Yaskawa INFORM job: R1_W45-48(90,0)KM-OK.JBI

/JOB
//NAME R1_W45-48(90,0)KM-OK
///FOLDERNAME KRIS-SCIANA
//POS
///NPOS 86,86,0,6,0,0
///TOOL 0
///POSTYPE PULSE
///PULSE
C00000=614,-36100,-109393,-1002,105622,76266
C00001=-30112,-127063,-118472,9266,74977,65479
C00002=-146783,-41222,-44528,14508,92298,23932
C00003=-177758,-18432,-24897,15900,96897,12902
C00004=-166847,35431,29185,16026,89350,15768
C00005=-166321,37118,32341,15327,88247,16677
C00006=-166321,37589,33997,15328,87496,16584
C00007=-166321,37118,32341,15327,88247,16677
C00008=-171699,4841,-760,15279,92918,15369
C00009=-170835,-35200,-22324,18799,58263,10772
C00010=-166066,-33100,-15421,17623,54185,12058
C00011=-165910,-32536,-14743,17588,54031,12098
C00012=-165593,-31712,-14199,17442,54048,12239
C00013=-167025,-37605,-22579,17571,56389,12034
C00014=-161139,-1958,-5557,939,83085,16350
C00015=-160390,25614,20531,865,81188,16590
C00016=-160390,25904,21696,866,80621,16587
C00017=-160640,27890,23636,893,80451,16499
C00018=-160390,25457,19886,865,81505,16593
C00019=-160390,25655,20697,865,81108,16591
C00020=-160390,25965,21925,866,80512,16587
C00021=-160390,25906,21695,866,80622,16587
C00022=-160724,27768,23517,901,80463,16471
C00023=-160390,25446,19834,865,81532,16594
C00024=-165643,13675,12551,10985,79337,20135
C00025=-167674,10013,12505,14753,77464,21361
C00026=-167674,10387,13747,14782,76911,21293
C00027=-167674,10317,13522,14776,77011,21304
C00028=-167700,12673,15637,14783,76929,21284
C00029=-167674,9804,11798,14735,77782,21397
C00030=-161667,10120,9793,4034,79193,25528
C00031=-160919,6459,2756,3926,81599,25861
C00032=-171280,-20527,-2481,28534,71438,-2255
C00033=-169873,-15007,4957,28696,69425,-2217
C00034=-167060,-14489,6711,28588,67760,-1526
C00035=-167060,-13749,8427,28718,67162,-1682
C00036=-167060,-14037,7762,28667,67393,-1622
C00037=-166465,-12361,9034,28595,67262,-1417
C00038=-167060,-14860,5838,28526,68066,-1445
C00039=-165078,-24102,-3856,28103,68483,-543
C00040=-174496,-24787,-5330,32767,69285,-4466
C00041=-172819,-19212,1769,32913,67371,-4356
C00042=-172173,-16914,4714,32988,66590,-4329
C00043=-171876,-16211,5234,32949,66511,-4228
C00044=-171876,-15504,6876,33099,65965,-4402
C00045=-171876,-15676,6480,33063,66097,-4360
C00046=-171337,-14366,7462,32993,65949,-4178
C00047=-171876,-15676,6480,33063,66097,-4360
C00048=-161265,-34405,-11426,23449,56557,2204
C00049=-165693,-30942,-7306,24884,57138,447
C00050=-166684,-37324,-14511,24847,58482,354
C00051=-186406,-34667,3928,73065,39460,38715
C00052=-184274,-31936,5659,72637,38187,39290
C00053=-183330,-31185,5556,72054,37725,39763
C00054=-184413,-32109,5553,72669,38270,39251
C00055=-183286,-31712,4384,71496,37848,40087
C00056=-183300,-30553,6129,72089,37695,39749
C00057=-184249,-31903,5681,72632,38172,39297
C00058=-186379,-34635,3948,73060,39445,38722
C00059=-168921,11501,9513,23787,62861,33812
C00060=-168977,15186,12854,23838,62728,33759
C00061=-168277,18170,15265,23592,62571,34011
C00062=-168933,14800,11613,23711,63235,33889
C00063=-168567,15646,14088,23805,62129,33795
C00064=-174514,12133,12884,25971,62948,31524
C00065=-174025,9736,7933,25443,64442,32081
C00066=-174066,6103,4745,25437,64541,32088
C00067=-165320,32292,30686,7449,75670,58759
C00068=-160580,40426,45052,9326,72009,60014
C00069=-168555,20447,28596,16427,68120,-19338
C00070=-168800,19872,28619,16504,67872,-19465
C00071=-157617,30618,37910,-7922,59943,61772
C00072=-157851,30496,37789,-7848,59932,61681
C00073=-159523,23474,32009,-7611,56187,61651
C00074=-170844,18084,26765,-2961,55783,56770
C00075=-171318,17827,26691,-2775,55680,56585
C00076=-172522,13662,24258,-755,52693,56042
C00077=-172766,11273,22657,-34,51599,55901
C00078=-172411,10671,22440,-198,51422,56051
C00079=-172687,-7816,-30,-66,55750,55932
C00080=-179212,-27838,-26858,-4490,80741,54483
C00081=-122151,-111635,-84959,-4490,80741,54483
C00082=-96954,-145656,-113562,11457,80138,54483
C00083=-72409,-164039,-132527,6736,11969,60674
C00084=-5263,-164039,-132527,6736,11969,60674
C00085=-5263,-164039,-132527,6736,-9043,60674
BC00000=262451,999,812332
BC00001=345212,1125,730788
BC00002=372391,1617,411462
BC00003=379607,1748,326684
BC00004=379648,1749,326197
BC00005=379648,1749,326197
BC00006=379648,1749,326197
BC00007=379648,1749,326197
BC00008=379648,1749,326197
BC00009=379648,1749,326197
BC00010=379648,1749,326197
BC00011=379648,1749,326197
BC00012=379648,1749,326197
BC00013=379648,1749,326197
BC00014=379648,1749,326197
BC00015=379648,1749,326197
BC00016=379648,1749,326197
BC00017=379648,1749,326197
BC00018=379648,1749,326197
BC00019=379648,1749,326197
BC00020=379648,1749,326197
BC00021=379648,1749,326197
BC00022=379648,1749,326197
BC00023=379648,1749,326197
BC00024=359715,496,350393
BC00025=352053,15,359694
BC00026=352053,15,359694
BC00027=352053,15,359694
BC00028=352053,15,359694
BC00029=352053,15,359694
BC00030=352053,15,359694
BC00031=352053,15,359694
BC00032=313868,15,405128
BC00033=313868,15,405128
BC00034=313868,15,405128
BC00035=313868,15,405128
BC00036=313868,15,405128
BC00037=313868,15,405128
BC00038=313868,15,405128
BC00039=313868,15,405128
BC00040=341595,15,387601
BC00041=341595,15,387601
BC00042=341595,15,387601
BC00043=341595,15,387601
BC00044=341595,15,387601
BC00045=341595,15,387601
BC00046=341595,15,387601
BC00047=341595,15,387601
BC00048=341595,15,387601
BC00049=341595,15,387601
BC00050=341595,15,387601
BC00051=380086,15,357591
BC00052=379357,15,337196
BC00053=379066,15,329038
BC00054=379066,15,329038
BC00055=379066,15,329038
BC00056=346528,15,329921
BC00057=346820,15,338079
BC00058=347549,15,358475
BC00059=398174,15,330978
BC00060=398174,15,307650
BC00061=398174,15,298319
BC00062=398174,15,298319
BC00063=398174,15,298319
BC00064=398174,15,298319
BC00065=398174,15,291055
BC00066=398174,15,314383
BC00067=396475,15,377766
BC00068=396475,15,377766
BC00069=376171,15,378238
BC00070=376171,15,378238
BC00071=396475,15,377766
BC00072=396475,15,377766
BC00073=396475,15,377766
BC00074=396475,15,377766
BC00075=396475,15,377766
BC00076=396475,15,377766
BC00077=396475,15,377766
BC00078=396475,15,377766
BC00079=396475,15,377766
BC00080=396476,15,377761
BC00081=396476,15,377761
BC00082=396476,15,998488
BC00083=342120,131,1013854
BC00084=4442,131,1013854
BC00085=4442,491441,1045653
///POSTYPE BASE
///RECTAN
///RCONF 0,0,0,0,1,0,0,0,0,0,0,0,0,0,0,0,0,0,0,0,0,0,0,0
P00006=2.006,1.622,-0.565,0.0000,0.0000,0.0000
///RCONF 0,0,0,0,0,0,0,0,0,0,0,0,0,0,0,0,0,0,0,0,0,0,0,0
P00023=-2.957,-4.083,2.762,0.0000,0.0000,0.0000
P00024=-1.466,-0.226,-0.419,0.0000,0.0000,0.0000
P00026=2.644,0.055,-2.583,0.0000,0.0000,0.0000
P00027=2.278,0.099,-4.210,0.0000,0.0000,0.0000
P00030=-0.014,-0.768,0.131,0.0000,0.0000,0.0000
//INST
///DATE 2024/09/16 12:08
///ATTR SC,RW
///GROUP1 RB1,BS1
NOP
'r1_W45-48(90,0)
'Path S904
SFTOF
MOVJ C00000 BC00000 VJ=100.00
MOVJ C00001 BC00001 VJ=100.00
MOVJ C00002 BC00002 VJ=100.00
MOVJ C00003 BC00003 VJ=100.00
MOVL C00004 BC00004 V=166.7
MOVL C00005 BC00005 V=60.0
REFP 3 C00006 BC00006
CALL JOB:SEARCH-R1
SET P026 P006
SFTON P026
MOVL C00007 BC00007 V=60.0
MOVL C00008 BC00008 V=133.3
MOVL C00009 BC00009 V=133.3
MOVL C00010 BC00010 V=133.3
MOVL C00011 BC00011 V=60.0
REFP 3 C00012 BC00012
CALL JOB:SEARCH-R1
SET P026 P006
SFTON P026
MOVL C00013 BC00013 V=100.0
MOVL C00014 BC00014 V=133.3
MOVL C00015 BC00015 V=100.0
MOVL C00016 BC00016 V=60.0
REFP 3 C00017 BC00017
CALL JOB:SEARCH-R1
SET P026 P006
SFTON P026
MOVL C00018 BC00018 V=60.0
'Path S902
SFTOF
MOVL C00019 BC00019 V=60.0
REFP 3 C00020 BC00020
CALL JOB:SEARCH-R1
SET P030 P006
SFTON P030
MOVL C00021 BC00021 V=60.0
REFP 3 C00022 BC00022
CALL JOB:SEARCH-R1
SET P030 P006
SFTON P030
MOVL C00023 BC00023 V=60.0
MOVL C00024 BC00024 V=166.7
MOVL C00025 BC00025 V=60.0
REFP 3 C00026 BC00026
CALL JOB:SEARCH-R1
SET P024 P006
SFTON P024
MOVL C00027 BC00027 V=60.0
REFP 3 C00028 BC00028
CALL JOB:SEARCH-R1
SET P024 P006
SFTON P024
MOVL C00029 BC00029 V=60.0
MOVL C00030 BC00030 V=166.7
MOVL C00031 BC00031 V=166.7
'Path S901
SFTOF
MOVJ C00032 BC00032 VJ=100.00
MOVJ C00033 BC00033 VJ=100.00
MOVL C00034 BC00034 V=60.0
REFP 3 C00035 BC00035
CALL JOB:SEARCH-R1
SET P023 P006
SFTON P023
MOVL C00036 BC00036 V=60.0
REFP 3 C00037 BC00037
CALL JOB:SEARCH-R1
SET P023 P006
SFTON P023
MOVL C00038 BC00038 V=60.0
MOVL C00039 BC00039 V=166.7
'Path S1151
SFTOF
MOVJ C00040 BC00040 VJ=100.00
MOVJ C00041 BC00041 VJ=100.00
MOVL C00042 BC00042 V=100.0
MOVL C00043 BC00043 V=60.0
REFP 3 C00044 BC00044
CALL JOB:SEARCH-R1
SET P027 P006
SFTON P027
MOVL C00045 BC00045 V=60.0
REFP 3 C00046 BC00046
CALL JOB:SEARCH-R1
SET P027 P006
SFTON P027
MOVL C00047 BC00047 V=60.0
MOVL C00048 BC00048 V=100.0
MOVL C00049 BC00049 V=166.7
MOVL C00050 BC00050 V=166.7
'Path W467
SFTOF
SFTON P027
CALL JOB:COFNIJ_DRUT
MOVJ C00051 BC00051 VJ=100.00
MOVJ C00052 BC00052 VJ=100.00
MOVL C00053 BC00053 V=100.0 PL=0
REFP 1 C00054 BC00054
REFP 2 C00055 BC00055
MACRO1 MJ#(0) ARGF9
ARCON
SFTON P023
MOVL C00056 BC00056 V=10.0
ARCOF
MOVL C00057 BC00057 V=166.7
MOVL C00058 BC00058 V=166.7
SFTOF
SFTON P026
MOVJ C00059 BC00059 VJ=100.00
MOVJ C00060 BC00060 VJ=100.00
MOVL C00061 BC00061 V=100.0 PL=0
REFP 1 C00062 BC00062
REFP 2 C00063 BC00063
MACRO1 MJ#(0) ARGF6
ARCON
WVON WEV#(40)
MOVL C00064 BC00064 V=7.5
ARCOF
WVOF
MOVL C00065 BC00065 V=166.7
MACRO1 MJ#(0) ARGF9
MOVL C00066 BC00066 V=166.7
SFTOF
'Path W474
SFTON P026
MOVJ C00067 BC00067 VJ=100.00
MOVL C00068 BC00068 V=100.0 PL=0
REFP 1 C00069 BC00069
REFP 2 C00070 BC00070
MACRO1 MJ#(0) ARGF6
ARCON
WVON WEV#(40)
MOVL C00071 BC00071 V=7.5
MOVL C00072 BC00072 V=7.5
WVOF
MACRO1 MJ#(0) ARGF9
SFTON P030
MOVL C00073 BC00073 V=10.0
SFTON P024
MOVL C00074 BC00074 V=10.0
MOVL C00075 BC00075 V=10.0
MOVL C00076 BC00076 V=10.0
MOVL C00077 BC00077 V=10.0
MOVL C00078 BC00078 V=10.0
ARCOF
SFTOF
MOVL C00079 BC00079 V=100.0
MOVL C00080 BC00080 V=166.7
MOVJ C00081 BC00081 VJ=100.00
MOVJ C00082 BC00082 VJ=100.00
MOVJ C00083 BC00083 VJ=100.00
MOVJ C00084 BC00084 VJ=100.00
MOVJ C00085 BC00085 VJ=100.00
SFTOF
END
